// TwinCAT 3 PLC project Server
// ProgramVersion: 3.1.0.9
// libraries:
//   VisuElem3DPath, 3.5.6.0 (System)
//   VisuElemMeter, 3.5.6.0 (System)
//   VisuElems, 3.5.6.10 (System)
//   VisuElemsDateTime, 3.5.6.0 (System)
//   VisuElemsSpecialControls, 3.5.6.0 (System)
//   VisuElemsWinControls, 3.5.6.0 (System)
//   VisuElemTextEditor, 3.5.6.0 (System)
//   visuinputs, 3.5.6.0 (system)
//   VisuNativeControl, 3.5.6.0 (System)
//   Tc2_EtherCAT, * (Beckhoff Automation GmbH)
//   Tc2_Standard, * (Beckhoff Automation GmbH)
//   Tc2_System, * (Beckhoff Automation GmbH)
//   Tc2_Utilities, * (Beckhoff Automation GmbH)
//   Tc3_Interfaces, * (Beckhoff Automation GmbH)
//   Tc3_Module, * (Beckhoff Automation GmbH)
// project tree:
//   DUTs/ TUhr.TcDUT
//   / GlobalTextList.TcGTLO, PlcTask.TcTTO, Visualisiserungsmanager.TcVMO (not stored)
//   GVLs/ GVL.TcGVL, GVL_Constants.TcGVL, GVL_Visu.TcGVL, Haus1.TcGVL, Haus2.TcGVL, Haus4.TcGVL, HausSim.TcGVL, Netzwerk.TcGVL
//   Images/ Icons.TcIPO (not stored), ImagePool.TcIPO (not stored)
//   POUs/ FB_Alarm_Bild.TcPOU, FB_Alarm.TcPOU, FB_Besucher.TcPOU, FB_DataHistory_Int.TcPOU, FB_DataHistory_Real.TcPOU, FB_Heizung.TcPOU, FB_Regenmacher.TcPOU, FB_Uhr.TcPOU, FB_Visu_BildToggle.TcPOU, FB_Wetterbericht.TcPOU, FB_Wind.TcPOU, GET_TIME.TcPOU, INT_R_TRIG.TcPOU, MAIN.TcPOU, FB_Sonne.TcPOU, PG_Besucher.TcPOU, PG_Sonne.TcPOU, PG_Heizung.TcPOU, PG_Regen.TcPOU, PG_Simulationshaus.TcPOU, PG_Time.TcPOU, PG_Alarm.TcPOU, INT_TRIG.TcPOU, PG_Wind.TcPOU, PG_Visu.TcPOU, Visu_Baum.TcPOU, Visu_DayNight.TcPOU
//   VISUs/ Haus_1.TcVIS, Haus_2.TcVIS, Haus_3.TcVIS, MainVisu.TcVIS, Simuliertes_Haus.TcVIS, Settings.TcVIS, Uhr.TcVIS, Wetterbericht.TcVIS, Zentrale.TcVIS
// real-time tasks:
//   TASK PlcTask: cycle T#10ms, priority 20, ADS port 350
// I/O:
//   DEVICE Netzvariablen (EtherCAT Automation Protocol) (disabled), AmsNetId 192.168.252.131.2.1
//     Server (Publisher)
//     Haus_01
//     Haus_02
//     Haus_04
// variable links:
//   Server/Server Instance <-> Netzvariablen (EtherCAT Automation Protocol)/Haus_01
//     PlcTask Inputs/Netzwerk.net_alarm_01 <-> net_alarm_01/Inputs/VarData
//     PlcTask Inputs/Netzwerk.net_besucher_01 <-> net_besucher_01/Inputs/VarData
//     PlcTask Inputs/Netzwerk.net_heizung_01 <-> net_heizung_01/Inputs/VarData
//     PlcTask Inputs/Netzwerk.net_licht_01 <-> net_licht_01/Inputs/VarData
//   Server/Server Instance <-> Netzvariablen (EtherCAT Automation Protocol)/Haus_02
//     PlcTask Inputs/Netzwerk.net_alarm_02 <-> net_alarm_02/Inputs/VarData
//     PlcTask Inputs/Netzwerk.net_besucher_02 <-> net_besucher_02/Inputs/VarData
//     PlcTask Inputs/Netzwerk.net_heizung_02 <-> net_heizung_02/Inputs/VarData
//     PlcTask Inputs/Netzwerk.net_licht_02 <-> net_licht_02/Inputs/VarData
//   Server/Server Instance <-> Netzvariablen (EtherCAT Automation Protocol)/Haus_04
//     PlcTask Inputs/Netzwerk.net_alarm_04 <-> net_alarm_04/Inputs/VarData
//     PlcTask Inputs/Netzwerk.net_besucher_04 <-> net_besucher_04/Inputs/VarData
//     PlcTask Inputs/Netzwerk.net_heizung_04 <-> net_heizung_04/Inputs/VarData
//     PlcTask Inputs/Netzwerk.net_licht_04 <-> net_licht_04/Inputs/VarData
//   Server/Server Instance <-> Netzvariablen (EtherCAT Automation Protocol)/Server (Publisher)
//     PlcTask Outputs/Netzwerk.net_einbruch_alarm <-> net_einbruch_alarm/Outputs/VarData
//     PlcTask Outputs/Netzwerk.net_heizung_out <-> net_heizung/Outputs/VarData
//     PlcTask Outputs/Netzwerk.net_regen <-> net_regen/Outputs/VarData
//     PlcTask Outputs/Netzwerk.net_reset_besucher <-> net_reset_besucher/Outputs/VarData
//     PlcTask Outputs/Netzwerk.net_sonne <-> net_sonne/Outputs/VarData
//     PlcTask Outputs/Netzwerk.net_wind <-> net_wind/Outputs/VarData

CONFIGURATION Server
    RESOURCE PLC ON TwinCAT3
        TASK PlcTask(INTERVAL := T#10ms, PRIORITY := 20);
        PROGRAM MAIN WITH PlcTask : MAIN;
    END_RESOURCE
END_CONFIGURATION

// ---- DUTs/TUhr.TcDUT
TYPE TUhr :
STRUCT
	Stunde : REAL;
	Minute : REAL;
	Sekunde : REAL;
END_STRUCT
END_TYPE

// ---- GVLs/GVL.TcGVL
VAR_GLOBAL
	Alarm_H1_V : BOOL;
	Alarm_H2_V : BOOL;
	Alarm_H4_V : BOOL;
	
	Licht : INT;
	Regen : BOOL;
	SimZeitMultiplikator : INT;
	RealtimeManipulator : INT := RealtimeManipulator_STD;

	SimTagesFortschritt : REAL;
	SimMilliSekunde : INT;
	SimSekunde : INT;
	SimMinute : INT;
	SimStunde : INT;
	
	RealMilliSekunde : INT;
	RealSekunde : INT;
	RealMinute : INT;
	RealStunde : INT;
	
	SimRealTagSeitStart : INT;
	RealTagSeitStart : INT;
	
	SonneHistory : ARRAY [0..DatenHistoryZaehler] OF INT;
	WindHistory : ARRAY [0..DatenHistoryZaehler] OF REAL;
	
	Wind_V : INT;
	Wind_Auto : BOOL;
	Wind_Auto_V : BOOL;
	BWind : BOOL;
	
	Sonne_Auto : BOOL;
	Sonne_Auto_V : BOOL;
	Sonne_V	: INT;
	Sonne_A	: INT;
	L_Sonnenstand : INT;
	L_Sonne : STRING;
	L_Himmel : DWORD;
	L_Baum : INT;
	
	GL_Besucher : INT;
	GL_Besucher_reset : BOOL;
	GL_Alarm_reset : BOOL;
	GL_Besucher_reset_A : BOOL;
	
	Regenwahrscheinlichkeit : INT := Regenwahrscheinlichkeit_STD;
END_VAR

// ---- GVLs/GVL_Constants.TcGVL
VAR_GLOBAL CONSTANT
	
	DatenHistoryZaehler : INT := 50;
	Licht_min : INT := 100;
	Licht_max : INT := 2500;
	Alarm_time : TIME := T#10S;
	Heizung_reaktion : TIME := T#20S;
	Maximum_Wind : REAL := 300;
	BildMond : STRING := 'Mond';
	BildSonne : STRING := 'Sonne';
	BildEinbruchAlarm : STRING := 'Einbruch_rot';
	BildEinbruchOk : STRING := 'Einbruch_grun';
	BildRegen : STRING := 'Regen';
	BildWolke : STRING := 'Wolke';
	BildLicht : STRING := 'Licht';
	BildDunkel : STRING := 'Dunkel';
	ICON_Mond : STRING := 'ICON_Mond';
	ICON_Sonne : STRING := 'ICON_Sonne';
	ICON_Wolke : STRING := 'ICON_Wolke';
	ICON_Regen : STRING := 'ICON_Regen';
	ICON_WindRegen : STRING := 'ICON_WindRegen';
	ICON_WindWolke : STRING := 'ICON_WindWolke';
	
	RealtimeManipulator_STD : INT := 0;	
	Regenwahrscheinlichkeit_STD : INT := 30;
	TagNachtFixGrad : INT := -90;
	TagNachtMaxTransparenz : INT := 255;
END_VAR

// ---- GVLs/GVL_Visu.TcGVL
VAR_GLOBAL
	Rege_Heute : BOOL;
	RegenSimStunde : INT;
	RegenSimMinute : INT;
	Regen_Dauer : INT;
	RegenSimStunde_Ende : INT;
	RegenSimMinute_Ende : INT;
	
	Wetterbericht_Bild : STRING;
	Wetterbericht_Vorhersage_Bild: STRING;
	
	Simulation : BOOL := FALSE;
	
	
	Uhr : TUhr;
	
END_VAR

// ---- GVLs/Haus1.TcGVL
VAR_GLOBAL
	// Einbruchbild
	L_EinbruchBild : STRING;
	// Bild der Wolke (Wetter)
	WetterBild : STRING := BildWolke;
	// Bild Licht (Im Haus)
	BildLicht : STRING := GVL_Constants.BildLicht;
END_VAR

// ---- GVLs/Haus2.TcGVL
VAR_GLOBAL
	L_EinbruchBild : STRING;
	WetterBild : STRING := BildWolke;
	BildLicht : STRING := GVL_Constants.BildLicht;
END_VAR

// ---- GVLs/Haus4.TcGVL
VAR_GLOBAL
	L_EinbruchBild : STRING;
	WetterBild : STRING := BildWolke;
	BildLicht : STRING := GVL_Constants.BildLicht;
END_VAR

// ---- GVLs/HausSim.TcGVL
VAR_GLOBAL
	// Licht brennt
	L_Licht : BOOL;
	// Licht einschalten (Visu)
	L_Licht_V : BOOL;
	// Einbruchbild (Wechset)
	L_EinbruchBild : STRING;
	// Bild der Wolke
	WetterBild : STRING := BildWolke;
	// Bild Licht im Haus
	BildLicht : STRING := GVL_Constants.BildLicht;
	
	// Besucher zähler
	Besucher : INT;
	// Hat alarm
	Alarm : BOOL;
	// Alarm eingeschalten
	Alarm_V : BOOL;
	// Heizung Simulation
	heizung_SIM : INT;
	
	// Klingeln (Visu)
	Sim_Haus_Glocke : BOOL;
	// Alarm einschalten (Visu)
	Sim_Haus_Alarm : BOOL;
	// Alarm zurücksetzen (Haus Visu)
	Sim_Haus_ResetAlarm: BOOL;
END_VAR

// ---- GVLs/Netzwerk.TcGVL
VAR_GLOBAL
// Licht im Haus 1
	net_licht_01 AT %I* : BOOL;
// Licht im Haus 2
	net_licht_02 AT %I* : BOOL;
// Licht im Haus 4
	net_licht_04 AT %I* : BOOL;
// Besucher im Haus 1
	net_besucher_01 AT %I* : INT;
// Besucher im Haus 2
	net_besucher_02 AT %I* : INT;
// Besucher im Haus 4
	net_besucher_04 AT %I* : INT;
// Alarm im Haus 1
	net_alarm_01 AT %I* : BOOL;
// Alarm im Haus 2
	net_alarm_02 AT %I* : BOOL;
// Alarm im Haus 4
	net_alarm_04 AT %I* : BOOL;
// Heizung im Haus 1
	net_heizung_01 AT %I* : INT;
// Heizung im Haus 2
	net_heizung_02 AT %I* : INT;
// Heizung im Haus 4
	net_heizung_04 AT %I* : INT;


// Globaler Alarm
	net_einbruch_alarm AT %Q* : BOOL;
// Globale Besucher reset
	net_reset_besucher AT %Q* : BOOL;
// Simulierter Wind
	net_wind AT %Q* : REAL;
// Simulierter Regen
	net_regen AT %Q* : BOOL;
// Simuliertes Licht
	net_sonne AT %Q* : REAL;
// Heizung resultat
	net_heizung_out AT %Q* : INT;
END_VAR

// ---- POUs/MAIN.TcPOU
PROGRAM MAIN
VAR
END_VAR

PG_Time();
PG_Alarm();
PG_Sonne();
PG_Regen();
PG_Heizung();
PG_Wind();
PG_Visu();
PG_Besucher();
PG_SimulationsHaus();

END_PROGRAM

// ---- POUs/PG_Time.TcPOU
PROGRAM PG_Time
VAR
	FAKE_TIME: GET_TIME;
	REAL_TIME: GET_TIME;
	FB_Uhr_0: FB_Uhr;
END_VAR

REAL_TIME(_speed := RealtimeManipulator); // GET_TIME
Fake_Time(_speed := SimZeitMultiplikator); // GET_TIME
SimTagesFortschritt := Fake_Time._prog;
RealMilliSekunde := REAL_TIME._ms;
SimMilliSekunde := Fake_Time._ms;
RealSekunde := REAL_TIME._s;
SimSekunde := Fake_Time._s;
RealMinute := REAL_TIME._m;
SimMinute := Fake_Time._m;
RealStunde := REAL_TIME._h;
SimStunde := Fake_Time._h;
RealTagSeitStart := REAL_TIME._days;
SimRealTagSeitStart := Fake_Time._days;
FB_Uhr_0(_h := SimStunde, _min := SimMinute, _s := SimSekunde); // FB_Uhr
Uhr.Stunde := FB_Uhr_0.deg_h;
Uhr.Minute := FB_Uhr_0.deg_min;
Uhr.Sekunde := FB_Uhr_0.deg_s;

END_PROGRAM

// ---- POUs/GET_TIME.TcPOU
FUNCTION_BLOCK GET_TIME
VAR_INPUT
	_speed : INT;
END_VAR
VAR_OUTPUT
	_prog : REAL;
	_ms : INT;
	_s : INT;
	_m : INT;
	_h : INT;
	_days : INT;
END_VAR
VAR
	systemTime : GETSYSTEMTIME;
	firstH : BOOL := TRUE;
	ms_count : UDINT;
END_VAR

// Systemzeit auslesen und in Millisekunden, Sekunden, Minuten, Stunden sowie den Tagesfrotschritt in % berechnen.
systemTime();
ms_count := systemTime.timeLoDW / 10000;
ms_count := ms_count * LREAL_TO_UDINT(EXPT(10, _speed));
_ms  := UDINT_TO_INT(ms_count MOD 1000);
_s := UDINT_TO_INT((ms_count / 1000) MOD 60);
_m := UDINT_TO_INT((ms_count / 60000) MOD 60); 
_h := UDINT_TO_INT(((ms_count / 3600000) MOD 24));
_prog := 360 * DINT_TO_REAL(_h * 3600000 + (_m+1) * 60000 + (_s+1) * 1000 + _ms) / UDINT_TO_REAL(24 * 3600000);

// Tage seit Systemstart zählen
IF _h MOD 24 = 0 THEN
	IF firstH THEN
		_days := _days + 1;
		firstH := FALSE;
	END_IF
ELSE
	firstH := TRUE;
END_IF

END_FUNCTION_BLOCK

// ---- POUs/FB_Uhr.TcPOU
FUNCTION_BLOCK FB_Uhr
VAR_INPUT
	_h : INT;
	_min : INT;
	_s : INT;
END_VAR
VAR_OUTPUT
	deg_h : REAL;
	deg_min : REAL;
	deg_s : REAL;
END_VAR
VAR
	History : ARRAY[0..2] OF INT;
END_VAR

IF History[0] <> _h THEN
	History[0] := _h;
	deg_h := 30 * _h;
END_IF
IF History[1] <> _min THEN
	History[1] := _min;
	deg_min := _min * 6;
END_IF
IF History[2] <> _s THEN
	History[2] := _s;
	deg_s := _s * 6;
END_IF

END_FUNCTION_BLOCK

// ---- POUs/PG_Alarm.TcPOU
PROGRAM PG_Alarm
VAR
	Alarm_Off_Time: TIME := GVL_CONSTANTS.Alarm_time;
	Alarm_0: FB_Alarm;
	Alarm_Bild: FB_Alarm_Bild;
END_VAR

Alarm_0(
    AL_H1 := net_alarm_01,
    AL_H1_V := Alarm_H1_V,
    AL_H2 := net_alarm_02,
    AL_H2_V := Alarm_H2_V,
    AL_H4 := net_alarm_04,
    AL_H4_V := Alarm_H4_V,
    Al_Sim := HausSim.Alarm,
    Simulation := Simulation,
    T_Alarm := Alarm_Off_Time,
    reset := GL_Alarm_reset); // FB_Alarm
net_einbruch_alarm := Alarm_0.GL_Alarm;
Alarm_Bild(
    alarm := net_einbruch_alarm,
    h1Alarm := net_alarm_01,
    h2Alarm := net_alarm_02,
    h4Alarm := net_alarm_04,
    hSimAlarm := HausSim.Alarm,
    Bild_Alarm := BildEinbruchAlarm,
    BIld_Ok := BildEinbruchOk); // FB_Alarm_Bild
Haus1.L_EinbruchBild := Alarm_Bild.SH1;
Haus2.L_EinbruchBild := Alarm_Bild.SH2;
Haus4.L_EinbruchBild := Alarm_Bild.SH4;
HausSim.L_EinbruchBild := Alarm_Bild.SHSim;

END_PROGRAM

// ---- POUs/FB_Alarm.TcPOU
FUNCTION_BLOCK FB_Alarm
VAR_INPUT
	AL_H1 : BOOL;	
	AL_H1_V : BOOL;
	AL_H2 : BOOL;
	AL_H2_V : BOOL;
	AL_H4 : BOOL;
	AL_H4_V : BOOL;
	Al_Sim : BOOL;
	Simulation : BOOL;
	T_Alarm : TIME;
	reset : BOOL;
END_VAR
VAR_OUTPUT
	GL_Alarm : BOOL;
END_VAR
VAR
	HatAlarm : BOOL;
	Alarm_On : TOF;
	Trig : F_TRIG;
	Alarm : RS;
END_VAR

IF Simulation THEN
HatAlarm := 
	AL_H1 OR 
	AL_H2 OR 
	AL_H4 OR 
	AL_H1_V OR 
	AL_H2_V OR 
	AL_H4_V OR
	AL_Sim;
ELSE
	HatAlarm := 
	AL_H1 OR 
	AL_H2 OR 
	AL_H4 OR 
	AL_H1_V OR 
	AL_H2_V OR 
	AL_H4_V;
END_IF
	
Alarm_On(IN := HatAlarm, PT := T_Alarm);
TRIG(CLK := Alarm_On.Q);
Alarm(SET := HatAlarm, RESET1 :=  TRIG.Q OR reset, Q1 => GL_Alarm);

END_FUNCTION_BLOCK

// ---- POUs/FB_Alarm_Bild.TcPOU
FUNCTION_BLOCK FB_Alarm_Bild
VAR_INPUT
	alarm : BOOL;
	h1Alarm : BOOL;
	h2Alarm : BOOL;
	h4Alarm : BOOL;
	hSimAlarm : BOOL;
	Bild_Alarm : STRING;
	BIld_Ok : STRING;
END_VAR
VAR_OUTPUT
	SH1 : STRING;
	SH2 : STRING;
	SH4 : STRING;
	SHSim : STRING;
END_VAR
VAR
	first : BOOL := TRUE;
	RTrig_H1 : R_TRIG;
	RTrig_H2 : R_TRIG;
	RTrig_H4 : R_TRIG;
	RTrig_HSim : R_TRIG;
	FTrig_H1 : F_TRIG;
	FTrig_H2 : F_TRIG;
	FTrig_h4 : F_TRIG;
	FTrig_HSim : F_TRIG;
END_VAR

RTrig_H1(CLK := h1Alarm);
FTrig_H1(CLK := h1Alarm);
RTrig_H2(CLK := h1Alarm);
FTrig_H2(CLK := h1Alarm);
RTrig_H4(CLK := h1Alarm);
FTrig_H4(CLK := h1Alarm);
FTrig_HSim(CLK := hSimAlarm);
RTrig_HSim(CLK := hSimAlarm);

IF first THEN
	IF h1Alarm THEN
		SH1 := Bild_Alarm;
	ELSE
		SH1 := Bild_Ok;
	END_IF
	IF h2Alarm THEN
		SH2 := Bild_Alarm;
	ELSE
		SH2 := Bild_Ok;
	END_IF
	IF h4Alarm THEN
		SH4 := Bild_Alarm;
	ELSE
		SH4 := Bild_Ok;
	END_IF
	IF hSimAlarm THEN
		SHSim := Bild_Alarm;
	ELSE
		SHSIM := Bild_Ok;
	END_IF
	
first := FALSE;

ELSE
	IF RTRIG_H1.Q THEN
		SH1 := Bild_Alarm;
	ELSIF FTRIG_H1.Q THEN
		SH1 := Bild_Ok;
	END_IF
	IF RTRIG_H2.Q THEN
		SH2 := Bild_Alarm;
	ELSIF FTRIG_H2.Q THEN
		SH2 := Bild_Ok;
	END_IF
	IF RTRIG_H4.Q THEN
		SH4 := Bild_Alarm;
	ELSIF FTRIG_H4.Q THEN
		SH4 := Bild_Ok;
	END_IF
	IF RTRIG_HSIM.Q THEN
		SHSIM := Bild_Alarm;
	ELSIF FTRIG_HSim.Q THEN
		SHSim := Bild_Ok;
	END_IF
END_IF

END_FUNCTION_BLOCK

// ---- POUs/PG_Sonne.TcPOU
PROGRAM PG_Sonne
VAR
	Sun_history: FB_DataHistory_Int;
	INT_TRIG_0: INT_TRIG;
	FB_Sonne_1: FB_Sonne;
	R_TRIG_0: R_TRIG;
END_VAR
VAR // added by the converter: edge detectors and wires of the graphical bodies
    _w1 : BOOL;
END_VAR

R_TRIG_0(CLK := Sonne_Auto_V); // R_TRIG
_w1 := R_TRIG_0.Q XOR _w1;
Sonne_Auto := NOT _w1;
FB_Sonne_1(
    _val := SimTagesFortschritt,
    _auto := Sonne_Auto,
    _visu_val := Sonne_V,
    _time := RealSekunde,
    _min := Licht_min,
    _max := Licht_max); // FB_Sonne
Licht := FB_Sonne_1._sin;
Sun_history(_val := FB_Sonne_1._sin, _save := FB_Sonne_1._trig); // FB_DataHistory_Int
SonneHistory := Sun_history._array;
net_sonne := REAL_TO_INT(Licht);

END_PROGRAM

// ---- POUs/FB_DataHistory_Int.TcPOU
FUNCTION_BLOCK FB_DataHistory_Int
VAR_INPUT
	_val : INT;
	_save : BOOL;
END_VAR
VAR_OUTPUT
	_array : ARRAY [0..DatenHistoryZaehler] OF INT;
END_VAR
VAR
	_i : INT;
END_VAR

IF _save THEN
	FOR _i := 0 TO DatenHistoryZaehler - 1 DO
		_array[_i] := _array[_i + 1];
	END_FOR
	_array[DatenHistoryZaehler] := _val;
END_IF

END_FUNCTION_BLOCK

// ---- POUs/INT_TRIG.TcPOU
FUNCTION_BLOCK INT_TRIG
VAR_INPUT
	_val : INT;
END_VAR
VAR_OUTPUT
	_Q : BOOL;
END_VAR
VAR
	History : INT;
	first : BOOL := TRUE;
END_VAR

// R_Trig und F_Trig in einem für INT Werte.
IF first THEN
	History := _val;
	first := FALSE;
ELSE
	IF History <> _val THEN
		_Q := TRUE;
		History := _val;
	ELSIF _Q THEN
		_Q := FALSE;	
	END_IF
END_IF

END_FUNCTION_BLOCK

// ---- POUs/FB_Sonne.TcPOU
FUNCTION_BLOCK FB_Sonne
VAR CONSTANT
	dayFix : INT := -90;
END_VAR
VAR_INPUT
	_val : REAL;
	_auto : BOOL;
	_visu_val : INT;
	_time : INT;
	_min : INT;
	_max : INT;
END_VAR
VAR_OUTPUT
	_sin : INT;
	_trig : BOOL;
END_VAR
VAR
	_do : BOOL;
	diff : INT;
	average : INT;
	T_Trig : INT_Trig;
END_VAR

// Trigger für die Ausführung alle 1sek.
T_Trig(_val := _time, _Q => _do);
// _do wird für die History (Statistik) verwendet.
_trig := _do;


// Wenn Licht Automatik eingeschalten, Automatisch berechnen
IF _do AND _auto THEN
	// Berechnen der Lichtemmission anhand der Uhrzeit _val
	diff := (_max - _min) / 2;
	average := REAL_TO_INT(_min + diff);
	_sin := LREAL_TO_INT(SIN(DEG_TO_RAD(_val + dayFix)) * diff + average);
ELSIF _do THEN
	// Wenn Licht Automatik ausgeschalten, Wert von Slider nehmen.
	_sin := _visu_val;
END_IF

END_FUNCTION_BLOCK

// ---- POUs/PG_Regen.TcPOU
PROGRAM PG_Regen
VAR
	Regenmacher: FB_Regenmacher;;
	Wetterbericht: FB_Wetterbericht;
END_VAR
VAR // added by the converter: edge detectors and wires of the graphical bodies
    _w1 : ANY;
END_VAR

Regenmacher(
    _gen := Regenwahrscheinlichkeit <> 0,
    _m := SimMinute,
    _h := SimStunde,
    _day := SimRealTagSeitStart,
    _prozent := Regenwahrscheinlichkeit,
    Simulation := TRUE); // FB_Regenmacher
Regen := Regenmacher._rain;
Rege_Heute := Regenmacher.HeuteRegen;
RegenSimStunde := Regenmacher.RegenStunde;
RegenSimMinute := Regenmacher.RegenMinute;
Regen_Dauer := Regenmacher.RegenDauer;
RegenSimStunde_Ende := Regenmacher.RegenBisStunde;
RegenSimMinute_Ende := Regenmacher.RegenBisMinute;
_w1 := SEL(Regen, BildWolke, BildRegen);
Haus1.WetterBild := _w1;
Haus2.WetterBild := _w1;
Haus4.WetterBild := _w1;
HausSim.WetterBild := _w1;
Wetterbericht(Regen := Regen, Wind := net_wind > 0); // FB_Wetterbericht
Wetterbericht_Bild := Wetterbericht.Aktuell;
Wetterbericht_Vorhersage_Bild := Wetterbericht.Vorhersage;

END_PROGRAM

// ---- POUs/FB_Regenmacher.TcPOU
FUNCTION_BLOCK FB_Regenmacher
VAR_INPUT
	_gen : BOOL;
	_m : INT;
	_h : INT;
	_day : INT;
	_prozent : INT;
	Simulation : BOOL;
END_VAR
VAR_OUTPUT
	_rain : BOOL;
	HeuteRegen : BOOL;
	RegenStunde : INT;
	RegenMinute : INT;
	RegenDauer : INT;
	RegenBisStunde : INT;
	RegenBisMinute : INT;
END_VAR
VAR
	dayTrig : INT_R_TRIG;
	RAND_H : DRAND;
	RAND_M : DRAND;
	RAND_D : DRAND;
END_VAR

IF _gen AND Simulation THEN
	dayTrig(_val := _day);
	
	IF dayTrig._Q THEN
		_rain := FALSE;
		HeuteRegen := FALSE;
		RAND_H(Seed := 0);
		HeuteRegen := LREAL_TO_INT(RAND_H.Num * 100) < _prozent;
		
		IF HeuteRegen THEN
			RAND_M(Seed := 1);
			RAND_D(Seed := 2);
			RegenStunde := LREAL_TO_INT(RAND_H.Num * 12);
			RegenMinute := LREAL_TO_INT(RAND_M.Num * 59);
			RegenDauer := LREAL_TO_INT(RAND_D.Num * 480);
			RegenBisStunde := RegenStunde + (RegenDauer / 60);
			RegenBisMinute := RegenMinute + (RegenDauer - ((RegenBisStunde - RegenStunde) * 60));
			IF RegenBisMinute > 60 THEN
				RegenBisStunde := RegenBisStunde + 1;
				RegenBisMinute := RegenBisMinute - 60;
			END_IF
		END_IF
	END_IF
	
	IF HeuteRegen THEN
		IF RegenStunde < _h OR (RegenStunde = _h AND RegenMinute <= _m) THEN
			_rain := TRUE;
			IF RegenBisStunde <= _h AND RegenBisMinute <= _m THEN
				_rain := FALSE;
				HeuteRegen := FALSE;
			END_IF
		END_IF
	END_IF
ELSE
	_rain := FALSE;
	HeuteRegen := FALSE;
END_IF

END_FUNCTION_BLOCK

// ---- POUs/INT_R_TRIG.TcPOU
FUNCTION_BLOCK INT_R_TRIG
VAR_INPUT
	_val : INT;
END_VAR
VAR_OUTPUT
	_Q : BOOL;
END_VAR
VAR
	History : INT;
	first : BOOL := TRUE;
END_VAR

// R_Trig für INT Werte. 
IF first THEN
	History := _val;
	first := FALSE;
ELSE
	IF History < _val THEN
		_Q := TRUE;
		History := _val;
	ELSIF _Q THEN
		_Q := FALSE;	
	END_IF
END_IF

END_FUNCTION_BLOCK

// ---- POUs/FB_Wetterbericht.TcPOU
FUNCTION_BLOCK FB_Wetterbericht
VAR_INPUT
	Regen : BOOL;
	Wind : BOOL;
	HeuteRegen : BOOL;
END_VAR
VAR_OUTPUT
	Aktuell : STRING;
	Vorhersage : STRING;
END_VAR
VAR
END_VAR

// Das richtige Icon anzeigen anhand der Wetterbedingungen
IF Regen AND Wind THEN
	Aktuell := GVL_CONSTANTS.ICON_WindRegen;
ELSIF Regen THEN
	Aktuell := GVL_CONSTANTS.ICON_Regen;
ELSIF Wind THEN
	Aktuell := GVL_CONSTANTS.ICON_WindWolke;
ELSE
	Aktuell := GVL_CONSTANTS.ICON_Wolke;
END_IF

IF HeuteRegen THEN
	Vorhersage := GVL_CONSTANTS.ICON_Regen;
ELSE
	Vorhersage := GVL_CONSTANTS.ICON_Wolke;
END_IF

END_FUNCTION_BLOCK

// ---- POUs/PG_Heizung.TcPOU
PROGRAM PG_Heizung
VAR
	FB_Heizung_0: FB_Heizung;
END_VAR

FB_Heizung_0(
    Heizung_01 := net_heizung_01,
    Heizung_02 := net_heizung_02,
    Heizung_04 := net_heizung_04,
    Heizung_Sim := HausSim.heizung_SIM,
    Simulation := Simulation,
    react := Heizung_reaktion); // FB_Heizung
net_heizung_out := FB_Heizung_0.Heizung;

END_PROGRAM

// ---- POUs/FB_Heizung.TcPOU
FUNCTION_BLOCK FB_Heizung
VAR_INPUT
	Heizung_01 : INT;
	Heizung_02 : INT;
	Heizung_04 : INT;
	Heizung_Sim : INT;
	Simulation : BOOL;
	react : TIME;
END_VAR
VAR_OUTPUT
	Heizung : INT;
END_VAR
VAR
	history : ARRAY [0..4] OF INT;
	first : BOOL := TRUE;
	_i : INT;
	maximum : INT := 0;
	timer : TON;
	
	run_timer : BOOL := FALSE;
END_VAR

IF FIRST THEN
	history[0] := Heizung_01;
	history[1] := Heizung_02;
	history[2] := Heizung_04;
	IF Simulation THEN
		history[3] := Heizung_Sim;
	ELSE
		history[3] := 0;
	END_IF
	
	FOR _i := 0 TO 3 DO
		IF history[_i] > maximum THEN
			maximum := history[_i];
		END_IF
	END_FOR
	history[4] := maximum;
	IF maximum < 15 THEN
		Heizung := 15;
	ELSIF maximum > 30 THEN
		Heizung := 30;
	ELSE
		Heizung := maximum;
	END_IF

	FIRST := FALSE;
ELSE
	// Wen es eine Änderung der Werte gab (Sim Haus nur miteinbeziehen, wenn Simulation eingeschalten ist.
	IF history[0] <> Heizung_01 OR history[1] <> Heizung_02 OR history[2] <> Heizung_04 OR (history[3] <> Heizung_Sim AND Simulation) THEN
		history[0] := Heizung_01;
		history[1] := Heizung_02;
		history[2] := Heizung_04;
		
		IF Simulation THEN
			history[3] := Heizung_Sim;
		ELSE
			history[3] := 0;
		END_IF
		
		// Höchsten Wert finden
		FOR _i := 0 TO 3 DO
			IF history[_i] > maximum THEN
				maximum := history[_i];
			END_IF
		END_FOR
		// Prüfen ob Wert ungleich beim Letzen mal und Timer starten bis neue Temperatur gesendet wird
		IF maximum <> history[4] THEN
			run_timer := TRUE;
			history[4] := maximum;	
		END_IF
	END_IF
END_IF

// Sendeverzögerung der neuen Temperatur.
IF run_timer THEN
	IF timer.Q THEN
		run_timer := FALSE;
		IF history[4] < 15 THEN
			Heizung := 15;
		ELSIF history[4] > 30 THEN
			Heizung := 30;
		ELSE
			Heizung := history[4];
		END_IF
	END_IF
	timer(IN := run_timer, PT := react);
END_IF

END_FUNCTION_BLOCK

// ---- POUs/PG_Wind.TcPOU
PROGRAM PG_Wind
VAR
	FB_Wind_0: FB_Wind;
	INT_TRIG_0: INT_TRIG;
	FB_DataHistory_Real_0: FB_DataHistory_Real;
	R_TRIG_0: R_TRIG;
END_VAR
VAR // added by the converter: edge detectors and wires of the graphical bodies
    _w1 : BOOL;
END_VAR

R_TRIG_0(CLK := Wind_Auto_V); // R_TRIG
_w1 := R_TRIG_0.Q XOR _w1;
Wind_Auto := NOT _w1;
FB_Wind_0(_auto := Wind_auto, _wind_V := Wind_V, _max := GVL_Constants.Maximum_Wind, _time := RealSekunde); // FB_Wind
net_wind := FB_Wind_0.Wind;
FB_DataHistory_Real_0(_val := FB_Wind_0.Wind, _save := FB_Wind_0.Trig); // FB_DataHistory_Real
WindHistory := FB_DataHistory_Real_0._array;
BWInd := net_wind > 0;

END_PROGRAM

// ---- POUs/FB_Wind.TcPOU
FUNCTION_BLOCK FB_Wind
VAR_INPUT
	_auto : BOOL;
	_wind_V : INT;
	_max : REAL;
	_time : INT;
END_VAR
VAR_OUTPUT
	Wind : REAL := 0;
	Trig : BOOL;
END_VAR
VAR
	Count : INT := 0;
	speed : REAL := 0.01;
	Step : BOOL := TRUE;
	valToAdd : REAL;
	
	StartTime : TON;
	StopTime : TON;
	NoWind : TP;
	NoWindFirst : BOOL := TRUE;
	StartT : TIME := T#2S;
	StopT : TIME := T#2S;
	Rand : DRAND;
	Direction : BOOL := TRUE;
	Prog : REAL;
	Height : REAL := 100;
	T_Trig : INT_Trig;
	_do : BOOL;
	_manipulator : INT := 100;
	WindToZero : REAL;
	BWindToZero : BOOL := FALSE;
 END_VAR

StartTime(IN := Direction, PT := StartT);
StopTime(IN := NOT Direction, PT := StopT);
T_TRIG(_val := _time, _Q => _do);
NoWind(IN := count = 0, PT := T#30S);

Trig := _do;

IF NoWind.Q THEN
	_do := FALSE;
	Wind := 0;
END_IF

IF _do AND _auto THEN
	IF Direction THEN
		Prog := ( TIME_TO_REAL(StartTime.ET) / TIME_TO_REAL(StartT) ) * 90 ;
		IF StartTime.Q THEN
			Direction := FALSE;
			Rand();
			StopT := LREAL_TO_TIME(Rand.Num * 10000);
			count := count + 1;
		END_IF
	ELSE
		IF count = 7 THEN
			WindToZero := Wind;
			BWindToZero := TRUE;
		END_IF
		
		Prog := 90 - ( TIME_TO_REAL(StopTime.ET) / TIME_TO_REAL(StopT) ) * 90;
		
		IF StopTime.Q THEN
				Direction := TRUE;
				Rand();
				StartT := LREAL_TO_TIME(Rand.Num * 10000);
				Step := NOT STEP;
				IF count = 7 THEN
					count := 0;
					BWindToZero := FALSE;
				ELSE
					count := count + 1;
				END_IF
			END_IF
	END_IF	

	IF count = 7 AND BWindToZero THEN
		Wind := WindToZero * LREAL_TO_REAL(SIN(DEG_TO_RAD(Prog)));
	ELSE
		valToAdd := LREAL_TO_REAL(SIN(DEG_TO_RAD(Prog)) * (TIME_TO_REAL(StartT) / _manipulator) ) ;
			
		IF STEP THEN
			valToAdd := valToAdd * ((_max - Wind) / _max);
			Wind := WIND + valToAdd;
		ELSE
			valToAdd := valToAdd * (Wind / _max);
			Wind := WIND - valToAdd;
		END_IF
	END_IF
END_IF

IF NOT _auto THEN
	Wind := _wind_V;
END_IF

END_FUNCTION_BLOCK

// ---- POUs/FB_DataHistory_Real.TcPOU
FUNCTION_BLOCK FB_DataHistory_Real
VAR_INPUT
	_val : REAL;
	_save : BOOL;
END_VAR
VAR_OUTPUT
	_array : ARRAY [0..DatenHistoryZaehler] OF REAL;
END_VAR
VAR
	_i : INT;
END_VAR

IF _save THEN
	FOR _i := 0 TO DatenHistoryZaehler - 1 DO
		_array[_i] := _array[_i + 1];
	END_FOR
	_array[DatenHistoryZaehler] := _val;
END_IF

END_FUNCTION_BLOCK

// ---- POUs/PG_Visu.TcPOU
PROGRAM PG_Visu
VAR
	Visu_Baum_0: Visu_Baum;
	INT_TRIG_0: INT_TRIG;
	Visu_DayNight_0: Visu_DayNight;
	INT_TRIG_1: INT_TRIG;
	BildToggle_Haus1: FB_Visu_BildToggle;
	BildToggle_Haus2: FB_Visu_BildToggle;
	BildToggle_Haus4: FB_Visu_BildToggle;
	BildToggle_HausSim: FB_Visu_BildToggle;
END_VAR
VAR // added by the converter: edge detectors and wires of the graphical bodies
    _w1 : ANY;
END_VAR

BildToggle_HausSim(val := HausSim.L_Licht, s_t := GVL_Constants.BildLicht, s_f := GVL_Constants.BildDunkel); // FB_Visu_BildToggle
BildToggle_Haus4(s_t := GVL_Constants.BildLicht, s_f := GVL_Constants.BildDunkel); // FB_Visu_BildToggle
Haus1.BildLicht := BildToggle_Haus1.BILD;
BildToggle_Haus2(val := net_licht_02, s_t := GVL_Constants.BildLicht, s_f := GVL_Constants.BildDunkel); // FB_Visu_BildToggle
INT_TRIG_1(_val := SimSekunde / 10); // INT_TRIG
Haus2.BildLicht := BildToggle_Haus2.BILD;
Haus4.BildLicht := BildToggle_Haus4.BILD;
HausSim.BildLicht := BildToggle_HausSim.BILD;
_w1 := (INT_TRIG_1._Q OR INT_TRIG_0._Q) AND BWind;
INT_TRIG_0(_val := SimMilliSekunde / 10); // INT_TRIG
Visu_Baum_0(_rotate := _w1, _speed := 1, _minDeg := -20, _maxDeg := 20); // Visu_Baum
L_Baum := Visu_Baum_0._rot;
Visu_DayNight_0(_deg := SimTagesFortschritt, licht := Licht, Licht_min := Licht_min, Licht_max := Licht_max); // Visu_DayNight
L_Sonne := Visu_DayNight_0._day;
L_Sonnenstand := Visu_DayNight_0._stand;
L_Himmel := Visu_DayNight_0._sun;
BildToggle_Haus1(val := net_licht_01, s_t := GVL_Constants.BildLicht, s_f := GVL_Constants.BildDunkel); // FB_Visu_BildToggle
// net_licht_04: input not connected

END_PROGRAM

// ---- POUs/Visu_Baum.TcPOU
FUNCTION_BLOCK Visu_Baum
VAR_INPUT
_rotate : BOOL;	
_speed : INT;
_minDeg : INT := -90;
_maxDeg : INT := 90;
END_VAR
VAR_OUTPUT
	_rot : INT := 0;
END_VAR
VAR
	counter : INT;
	rotateRight : BOOL;
END_VAR

// Wenn es Windet, bewegt sich der Baum.
IF _rotate THEN
	IF rotateRight THEN
		IF _rot > _maxDeg THEN
			rotateRight := FALSE;
		ELSE
			_rot := _rot + _speed;
		END_IF
	ELSE
		IF _rot < _minDeg THEN
			rotateRight := TRUE;
		ELSE
			_rot := _rot - _speed;
		END_IF
	END_IF
END_IF

END_FUNCTION_BLOCK

// ---- POUs/Visu_DayNight.TcPOU
FUNCTION_BLOCK Visu_DayNight
VAR CONSTANT
	Fix_Degree : INT := GVL_Constants.TagNachtFixGrad;
END_VAR
VAR_INPUT
	_deg : REAL;
	licht : INT;
	Licht_min : INT;
	Licht_max : INT;
END_VAR
VAR_OUTPUT
	_day : STRING;
	_stand : INT;
	_sun : DWORD;
END_VAR
VAR
	timeProg : REAL;
	transparency : INT := GVL_Constants.TagNachtMaxTransparenz;
	color : STRING;
	HEX : STRING;
END_VAR

timeProg := _deg + Fix_Degree;
IF timeProg < 0 OR timeProg > 180 THEN
	_stand := REAL_TO_INT(timeProg + 180);
	_day := GVL_Constants.BildMond;
ELSE
	_day := GVL_Constants.BildSonne;
	_stand := REAL_TO_INT(timeProg);
END_IF

transparency := REAL_TO_INT( ((Licht - Licht_min) / INT_TO_REAL(Licht_max - Licht_min)) * GVL_Constants.TagNachtMaxTransparenz );

HEX := DWORD_TO_HEXSTR(INT_TO_UINT(transparency), 2, FALSE);

color := '16#';
color := CONCAT(color, HEX);
color := CONCAT(color, 'FFFF00');

_sun := STRING_TO_DWORD(color);

END_FUNCTION_BLOCK

// ---- POUs/FB_Visu_BildToggle.TcPOU
FUNCTION_BLOCK FB_Visu_BildToggle
VAR_INPUT
	val : BOOL;
	s_t : STRING;
	s_f : STRING;
END_VAR
VAR_OUTPUT
	BILD : STRING;
END_VAR
VAR
	FIRST : BOOL := TRUE;
	history : BOOL;
END_VAR

// Selectorbaustein um einen String (Bild ID) Zumzuschalten
IF FIRST THEN
	IF val THEN
		BILD := s_t;
	ELSE
		BILD := s_f;
	END_IF
	history := val;
END_IF

IF val <> history THEN
	IF val THEN
		BILD := s_t;
	ELSE
		BILD := s_f;
	END_IF
	history := val;
END_IF

END_FUNCTION_BLOCK

// ---- POUs/PG_Besucher.TcPOU
PROGRAM PG_Besucher
VAR
	FB_Besucher_0: FB_Besucher;
	INT_R_TRIG_0: INT_R_TRIG;
END_VAR

INT_R_TRIG_0(_val := SimRealTagSeitStart); // INT_R_TRIG
GL_Besucher_reset_A := INT_R_TRIG_0._Q;
FB_Besucher_0(
    bes_H1 := net_besucher_01,
    bes_H2 := net_besucher_02,
    bes_H4 := net_besucher_04,
    bes_Sim := HausSim.Besucher,
    Simulation := Simulation,
    res_V := GL_Besucher_reset,
    res_A := GL_Besucher_reset_A); // FB_Besucher
GL_Besucher := FB_Besucher_0.besucher;
net_reset_besucher := FB_Besucher_0.res;

END_PROGRAM

// ---- POUs/FB_Besucher.TcPOU
FUNCTION_BLOCK FB_Besucher
VAR_INPUT
	bes_H1 : INT;
	bes_H2 : INT;
	bes_H4 : INT;
	bes_Sim : INT;
	Simulation : BOOL;
	res_V : BOOL;
	res_A : BOOL;
END_VAR
VAR_OUTPUT
	besucher : INT;
	res : BOOL;
END_VAR
VAR
END_VAR

IF Simulation THEN
	besucher := bes_H1 + bes_H2 + bes_H4 + bes_Sim;
ELSE
	besucher := bes_H1 + bes_H2 + bes_H4;
END_IF
IF res_V OR res_A THEN
	res := TRUE;
ELSE
	res := FALSE;
END_IF

END_FUNCTION_BLOCK

// ---- POUs/PG_Simulationshaus.TcPOU
PROGRAM PG_Simulationshaus
VAR
	Besucher: CTU;
	RS_0: RS;
	R_TRIG_0: R_TRIG;
	R_TRIG_1: R_TRIG;
END_VAR
VAR // added by the converter: edge detectors and wires of the graphical bodies
    _w1, _w2 : BOOL;
END_VAR

Besucher(CU := Sim_Haus_Glocke, RESET := net_reset_besucher); // CTU
HausSim.Besucher := WORD_TO_INT(Besucher.CV);
R_TRIG_0(CLK := HausSim.Alarm_V); // R_TRIG
_w1 := R_TRIG_0.Q XOR _w1;
HausSim.Alarm := _w1;
R_TRIG_1(CLK := HausSim.L_Licht_V); // R_TRIG
_w2 := R_TRIG_1.Q XOR _w2;
HausSim.L_Licht := _w2;

END_PROGRAM

// ---- GlobalTextList.TcGTLO
TEXTLIST GlobalTextList
  68 = ''
  26 = '%10i'
  15 = '%10s'
  1 = '%2f'
  2 = '%2i'
  4 = '%2i : '
  3 = '%2i : %2i : %2i'
  13 = '%2i Lumen'
  28 = '%2i Regenwahrscheinlichkeit'
  11 = '%2i Tage '
  10 = '%2i Tge '
  9 = '%2ih'
  8 = '%2imin'
  6 = '%2ims'
  7 = '%2is'
  62 = '%2r km/h Wind'
  5 = '%i'
  30 = '%i %'
  51 = '%i : Heizung'
  63 = '%i km/h Wind'
  66 = '%i Lumen'
  29 = '%i Regenwahrscheinlichkeit'
  14 = '%s'
  37 = 'Aktuelles Wetter'
  18 = 'Alarm'
  21 = 'Alarm %b'
  57 = 'Alarm zurücksetzen'
  67 = 'asdf'
  16 = 'Besucher'
  17 = 'Besucher Hochzählen'
  56 = 'Besucher zurücksetzen'
  55 = 'Besucher zurücksetzen%i'
  22 = 'Besucher: %i'
  54 = 'Besucher: %i°C'
  20 = 'Besuchern'
  48 = 'Den ganzen Tag schönes Wetter'
  35 = 'Einstellungen'
  50 = 'Globaler Alarm'
  31 = 'Haus 1'
  32 = 'Haus 2'
  33 = 'Haus 4'
  19 = 'Heizung'
  24 = 'Heizung: %2i'
  25 = 'Heizung: %2r'
  23 = 'Heizung: %i'
  52 = 'Heizung: %i°C'
  59 = 'Licht'
  12 = 'Real Time'
  45 = 'Regen bis: %i'
  49 = 'Regen Dauer: %i'
  69 = 'Regen Dauer: %i min'
  41 = 'Regen um: %i'
  42 = 'Regen um: %i Uhr'
  27 = 'Regenwahrscheinlichkeit'
  36 = 'Schliessen'
  47 = 'Schön bis: %i'
  34 = 'Settings'
  60 = 'Simulation'
  58 = 'Simulations Haus'
  64 = 'Sonne'
  65 = 'Sonne Manuell'
  46 = 'Uhr %i'
  44 = 'Uhr und %i Minuten'
  43 = 'und %i Minuten'
  38 = 'Vorhersage'
  39 = 'Vorhersage  Heute'
  40 = 'Vorhersage Heute'
  61 = 'Wind Manuell'
  53 = 'Wind: %i'
  0 = 'Zeit Manipulation'
END_TEXTLIST

// ---- VISUs/Haus_1.TcVIS
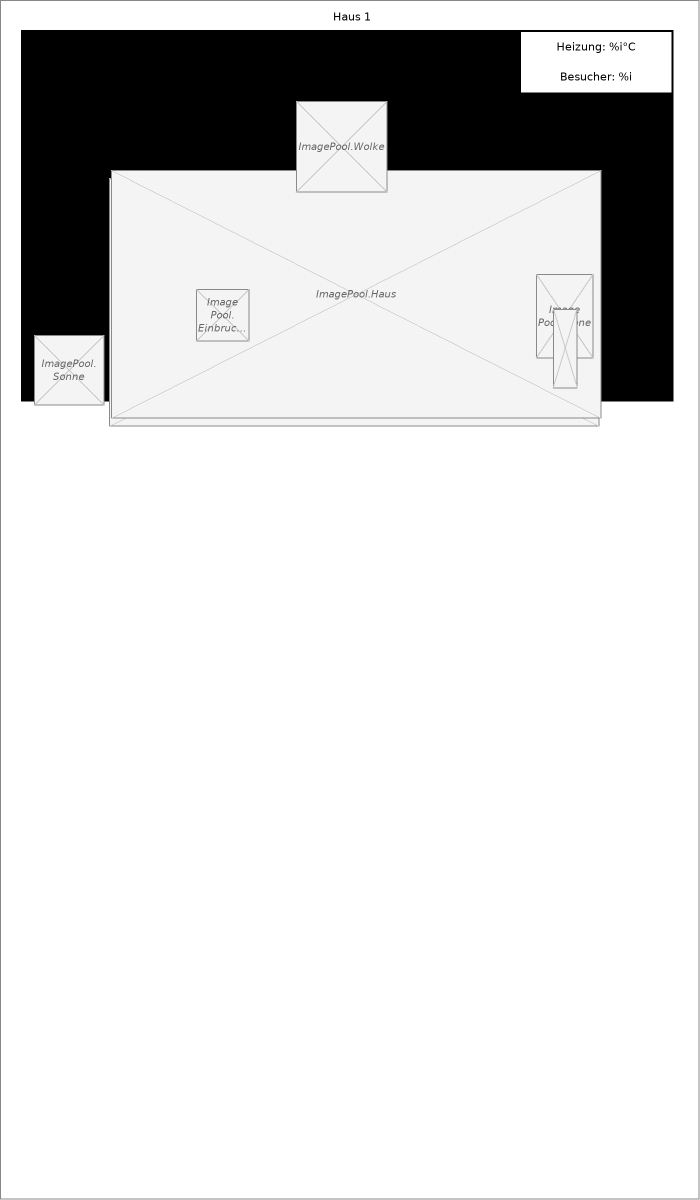
VISUALIZATION Haus_1  // 700x1200
    Rectangle (21,30 652x371)
    Rectangle (21,30 652x371), colour variable: L_Himmel
        p2167032090: L_Himmel
    Image (109,178 490x248), image: ImagePool.Licht
        p84334746: Haus1.BildLicht
    Image (111,170 490x248), image: ImagePool.Haus
    Image (536,274 57x84), image: ImagePool.Krone
        p2858320360: L_Baum
    Image (553,309 24x79), image: ImagePool.Stamm
    Image (34,335 70x70), image: ImagePool.Sonne
        p2858320360: L_Sonnenstand
        p84334746: L_Sonne
    Image (196,289 53x52), image: ImagePool.Einbruch_grun
        p84334746: Haus1.L_EinbruchBild
    Image (296,101 91x91), image: ImagePool.Wolke
        p84334746: Haus1.WetterBild
    Textfield (277,6 150x22), "Haus 1"
    Textfield (521,32 150x30), "Heizung: %i°C", text variable: net_heizung_01
    Textfield (521,62 150x30), "Besucher: %i", text variable: net_besucher_01
END_VISUALIZATION

// ---- VISUs/Haus_2.TcVIS
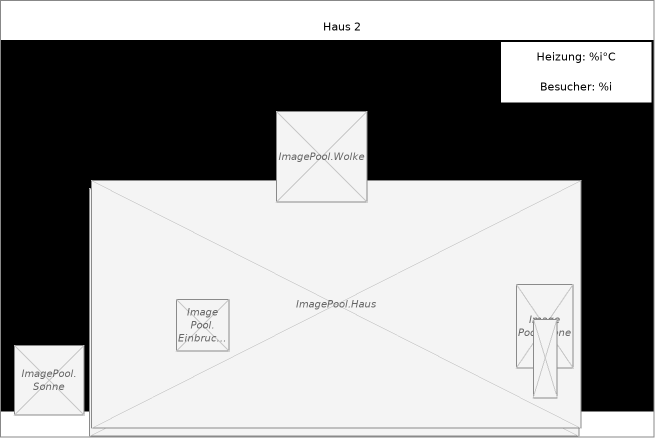
VISUALIZATION Haus_2  // 655x438
    Rectangle (1,40 652x371)
    Rectangle (1,40 652x371), colour variable: L_Himmel
        p2167032090: L_Himmel
    Image (89,188 490x248), image: ImagePool.Licht
        p84334746: Haus2.BildLicht
    Image (91,180 490x248), image: ImagePool.Haus
    Image (516,284 57x84), image: ImagePool.Krone
        p2858320360: L_Baum
    Image (533,319 24x79), image: ImagePool.Stamm
    Image (14,345 70x70), image: ImagePool.Sonne
        p2858320360: L_Sonnenstand
        p84334746: L_Sonne
    Image (176,299 53x52), image: ImagePool.Einbruch_grun
        p84334746: Haus2.L_EinbruchBild
    Image (276,111 91x91), image: ImagePool.Wolke
        p84334746: Haus2.WetterBild
    Textfield (267,16 150x22), "Haus 2"
    Textfield (501,42 150x30), "Heizung: %i°C", text variable: net_heizung_02
    Textfield (501,72 150x30), "Besucher: %i", text variable: net_besucher_02
END_VISUALIZATION

// ---- VISUs/Haus_3.TcVIS
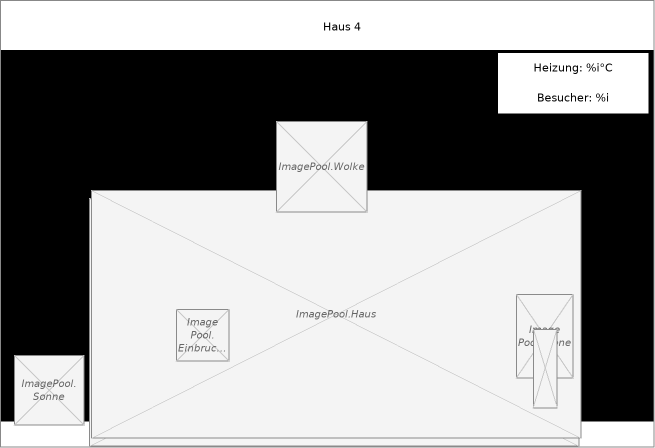
VISUALIZATION Haus_3  // 655x448
    Rectangle (1,50 652x371)
    Rectangle (1,50 652x371), colour variable: L_Himmel
        p2167032090: L_Himmel
    Image (89,198 490x248), image: ImagePool.Licht
        p84334746: Haus4.BildLicht
    Image (91,190 490x248), image: ImagePool.Haus
    Image (516,294 57x84), image: ImagePool.Krone
        p2858320360: L_Baum
    Image (533,329 24x79), image: ImagePool.Stamm
    Image (14,355 70x70), image: ImagePool.Sonne
        p2858320360: L_Sonnenstand
        p84334746: L_Sonne
    Image (176,309 53x52), image: ImagePool.Einbruch_grun
        p84334746: Haus4.L_EinbruchBild
    Image (276,121 91x91), image: ImagePool.Wolke
        p84334746: Haus4.WetterBild
    Textfield (267,16 150x22), "Haus 4"
    Textfield (498,53 150x30), "Heizung: %i°C", text variable: net_heizung_04
    Textfield (498,83 150x30), "Besucher: %i", text variable: net_besucher_04
END_VISUALIZATION

// ---- VISUs/MainVisu.TcVIS
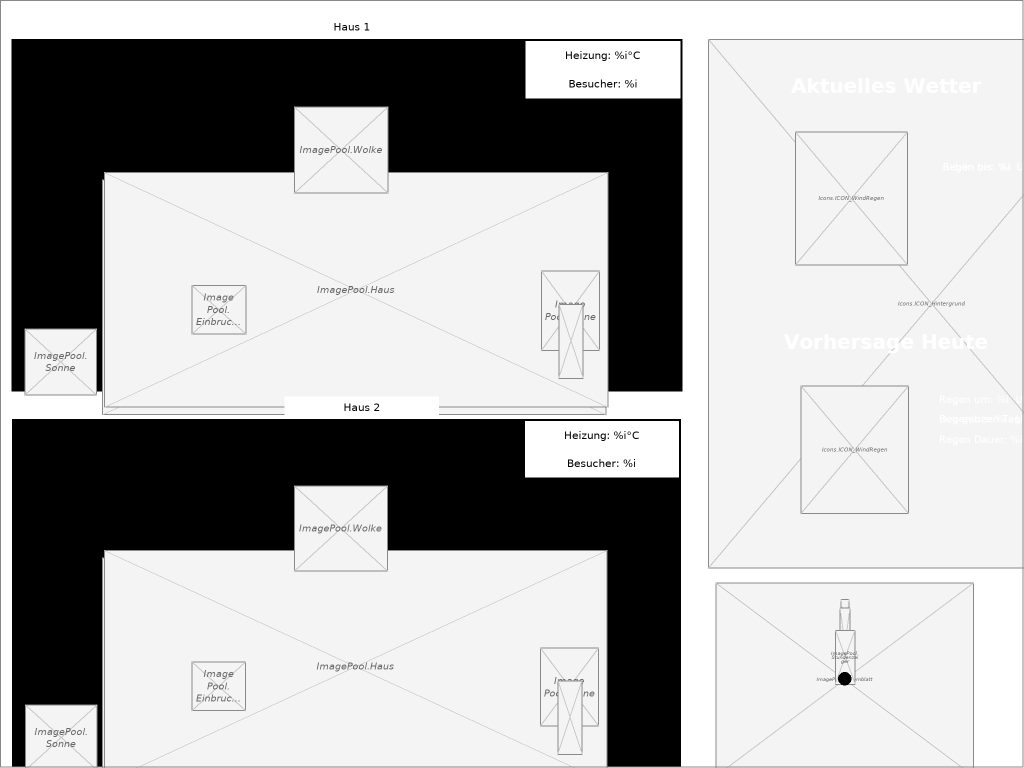
VISUALIZATION MainVisu  // 1024x768
    Frame (-10,11 720x1138), frame switch variable: Simulation
        shows Haus_1()
        shows Simuliertes_Haus()
    Frame (8,754 678x410), invisible if: Simulation
        shows Haus_3()
    Frame (11,382 672x410), invisible if: Simulation
        shows Haus_2()
    Button (1325,51 150x30), "Settings"
        OnMouseClick: OpenDialog Dialog=Settings, OpenModal=True, OpenCentered=True
    Frame (709,39 572x508)
        shows Wetterbericht()
    Frame (713,819 291x209)
        shows Zentrale()
    Button (1327,112 150x30), "Simulation"
        toggle Simulation
        OnMouseClick: OpenDialog Dialog=Simuliertes_Haus, OpenModal=True, PositionX=50, PositionY=50
        OnMouseClick: CloseDialog Dialog=Simuliertes_Haus, Result=OK, NumpadKeypadSet=True
    Frame (736,574 226x226)
        shows Uhr()
END_VISUALIZATION

// ---- VISUs/Simuliertes_Haus.TcVIS
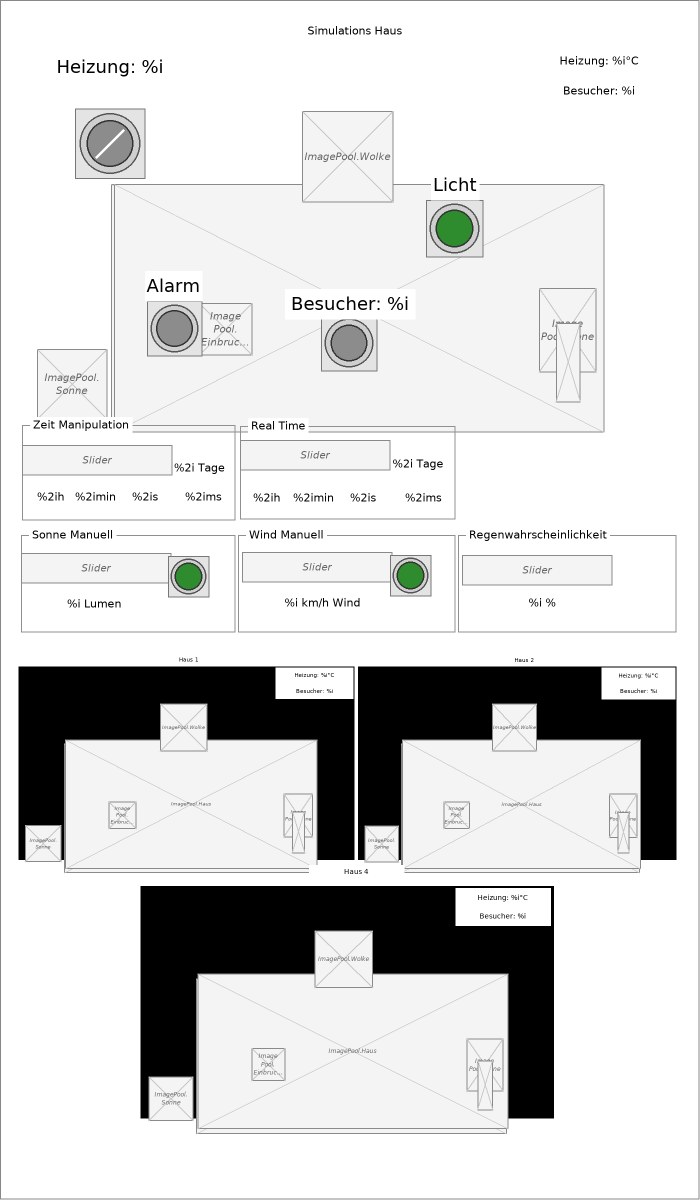
VISUALIZATION Simuliertes_Haus  // 700x1200
    Frame (8,651 360x625)
        shows Haus_1()
    Rectangle (24,44 652x371)
    Rectangle (24,44 652x371), colour variable: L_Himmel
        p2167032090: L_Himmel
    Image (111,184 490x248), image: ImagePool.Licht
        p84334746: HausSim.BildLicht
    Image (114,184 490x248), image: ImagePool.Haus
    Image (539,288 57x84), image: ImagePool.Krone
        p2858320360: L_Baum
    Image (556,323 24x79), image: ImagePool.Stamm
    Image (37,349 70x70), image: ImagePool.Sonne
        p2858320360: L_Sonnenstand
        p84334746: L_Sonne
    Image (199,303 53x52), image: ImagePool.Einbruch_grun
        p84334746: HausSim.L_EinbruchBild
    Image (302,111 91x91), image: ImagePool.Wolke
        p84334746: HausSim.WetterBild
    PushSwitch (147,300 55x57), variable: HausSim.Alarm_V, behaviour: TAP, style: Switch-PushSwitch-Gray
    Rectangle (145,271 57x30), "Alarm"
    Textfield (280,20 150x22), "Simulations Haus"
    Textfield (524,46 150x30), "Heizung: %i°C", text variable: HausSim.heizung_SIM
    Textfield (524,76 150x30), "Besucher: %i", text variable: HausSim.Besucher
    GroupBox (22,417 213x103), "Zeit Manipulation"
        Slider (0,28 150x30), variable: SimZeitMultiplikator, scale 0..4
        Textfield (41,65 65x30), "%2imin", text variable: SimMinute
        Textfield (90,65 66x30), "%2is", text variable: SimSekunde
        Textfield (148,65 67x30), "%2ims", text variable: SimMilliSekunde
        Textfield (-2,65 62x30), "%2ih", text variable: SimStunde
        Textfield (149,36 61x30), "%2i Tage", text variable: SimRealTagSeitStart
    PushSwitch (426,200 57x57), variable: HausSim.L_Licht_V, behaviour: TAP, style: Switch-PushSwitch-Green
    Rectangle (431,170 48x30), "Licht", text variable: HausSim.Besucher
    GroupBox (240,418 215x101), "Real Time"
        Textfield (149,31 62x30), "%2i Tage", text variable: RealTagSeitStart
        Slider (0,22 150x30), variable: RealtimeManipulator, scale 0..3
        Textfield (41,65 65x30), "%2imin", text variable: RealMinute
        Textfield (90,65 66x30), "%2is", text variable: RealSekunde
        Textfield (150,65 67x30), "%2ims", text variable: RealMilliSekunde
        Textfield (-4,65 62x30), "%2ih", text variable: RealStunde
    GroupBox (458,527 218x105), "Regenwahrscheinlichkeit"
        Slider (4,28 150x30), variable: Regenwahrscheinlichkeit, scale 0..100
        Textfield (-18,61 205x30), "%i %", text variable: Regenwahrscheinlichkeit
    GroupBox (238,527 217x105), "Wind Manuell"
        Slider (4,25 150x30), variable: Wind_V, scale 0..200
        Textfield (-18,61 205x30), "%i km/h Wind", text variable: net_wind
        PushSwitch (152,28 41x41), variable: Wind_Auto_V, behaviour: TAP, style: Switch-PushSwitch-Green
    GroupBox (21,527 214x105), "Sonne Manuell"
        Slider (0,26 150x30), variable: Sonne_V, scale 100..2500
        Textfield (4,62 139x30), "%i Lumen", text variable: net_sonne
        PushSwitch (147,29 41x41), variable: Sonne_Auto_V, behaviour: TAP, style: Switch-PushSwitch-Green
    Frame (358,646 319x228)
        shows Haus_2()
    Frame (140,855 415x280)
        shows Haus_3()
    PushSwitch (321,314 56x58), variable: Sim_Haus_Glocke, behaviour: TAP, style: Switch-PushSwitch-Gray
    Rectangle (285,289 130x30), "Besucher: %i", text variable: HausSim.Besucher
    Potentiometer360 (75,105 70x77), variable: heizung_SIM, style: Potentiometer-Potentiometer360-Gray, scale format: %.1f, scale 14..30
    Rectangle (35,52 150x30), "Heizung: %i", text variable: heizung_SIM
END_VISUALIZATION

// ---- VISUs/Settings.TcVIS
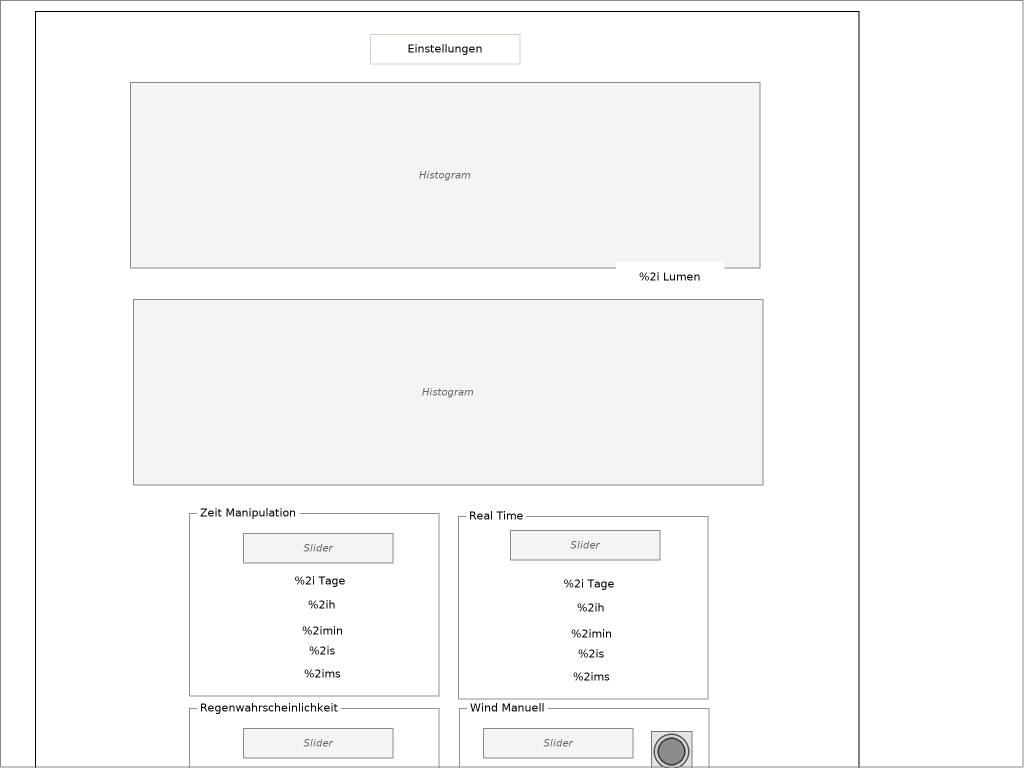
VISUALIZATION Settings  // 1024x768
    Rectangle (35,11 824x973)
    Histogram (130,82 630x186), scale format: %i, scale 0..3000
        p1518820177: SonneHistory
        p102497268: SonneHistory
        p788070771: ARRAY [0..DatenHistoryZaehler] OF INT
    GroupBox (189,505 250x191), "Zeit Manipulation"
        Slider (54,28 150x30), variable: SimZeitMultiplikator, scale 0..4
        Textfield (102,61 62x30), "%2i Tage", text variable: SimRealTagSeitStart
        Textfield (101,111 65x30), "%2imin", text variable: SimMinute
        Textfield (100,131 66x30), "%2is", text variable: SimSekunde
        Textfield (100,154 67x30), "%2ims", text variable: SimMilliSekunde
        Textfield (102,85 62x30), "%2ih", text variable: SimStunde
    GroupBox (458,508 250x191), "Real Time"
        Textfield (102,61 62x30), "%2i Tage", text variable: RealTagSeitStart
        Slider (52,22 150x30), variable: RealtimeManipulator, scale 0..3
        Textfield (101,111 65x30), "%2imin", text variable: RealMinute
        Textfield (100,131 66x30), "%2is", text variable: RealSekunde
        Textfield (100,154 67x30), "%2ims", text variable: RealMilliSekunde
        Textfield (102,85 62x30), "%2ih", text variable: RealStunde
    Textfield (616,262 108x30), "%2i Lumen", text variable: Licht
    GroupBox (189,700 250x105), "Regenwahrscheinlichkeit"
        Slider (54,28 150x30), variable: Regenwahrscheinlichkeit, scale 0..100
        Textfield (32,61 205x30), "%i %", text variable: Regenwahrscheinlichkeit
    Textfield (370,34 150x30), "Einstellungen"
    Button (680,929 150x30), "Schliessen"
        OnMouseClick: CloseDialog Dialog=Settings, Result=OK, NumpadKeypadSet=True
    Histogram (133,299 630x186), scale format: %i, scale 0..500
        p1518820177: WindHistory
        p102497268: WindHistory
        p788070771: ARRAY [0..DatenHistoryZaehler] OF REAL
    GroupBox (459,700 250x105), "Wind Manuell"
        Slider (24,28 150x30), variable: Wind_V, scale 0..200
        Textfield (2,61 205x30), "%i km/h Wind", text variable: net_wind
        PushSwitch (192,31 41x41), variable: Wind_Auto_V, behaviour: TAP, style: Switch-PushSwitch-Gray
    GroupBox (189,816 250x105), "Sonne Manuell"
        Slider (40,28 150x30), variable: Sonne_V, scale 100..2500
        Textfield (44,65 139x30), "%i Lumen", text variable: net_sonne
        PushSwitch (197,32 41x41), variable: Sonne_Auto_V, behaviour: TAP, style: Switch-PushSwitch-Gray
END_VISUALIZATION

// ---- VISUs/Uhr.TcVIS
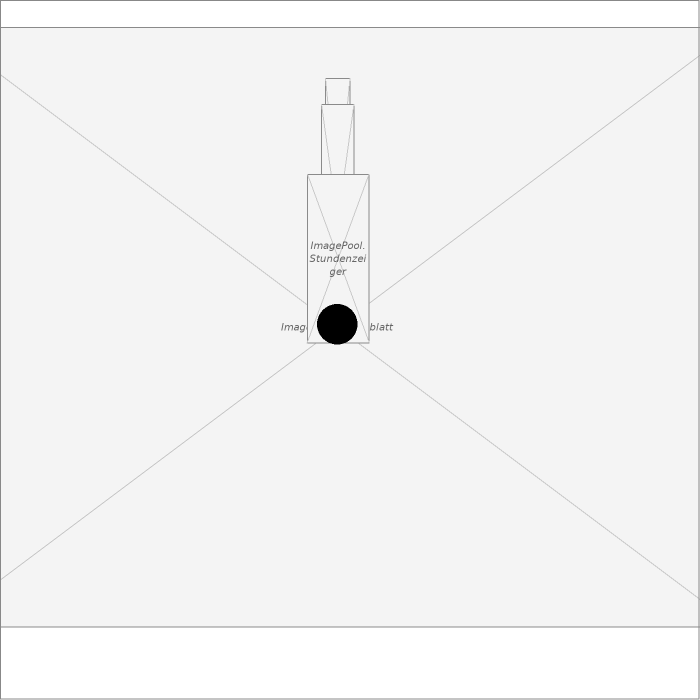
VISUALIZATION Uhr  // 700x700
    Image (-63,27 800x600), image: ImagePool.Ziffernblatt
    Image (325,78 25x260), image: ImagePool.Sekundenzeiger
        p2858320360: Uhr.Sekunde
    Image (321,104 33x239), image: ImagePool.Minutenzeiger
        p2858320360: Uhr.Minute
    Image (307,174 62x169), image: ImagePool.Stundenzeiger
        p2858320360: Uhr.Stunde
    Ellipse (317,304 40x40)
END_VISUALIZATION

// ---- VISUs/Wetterbericht.TcVIS
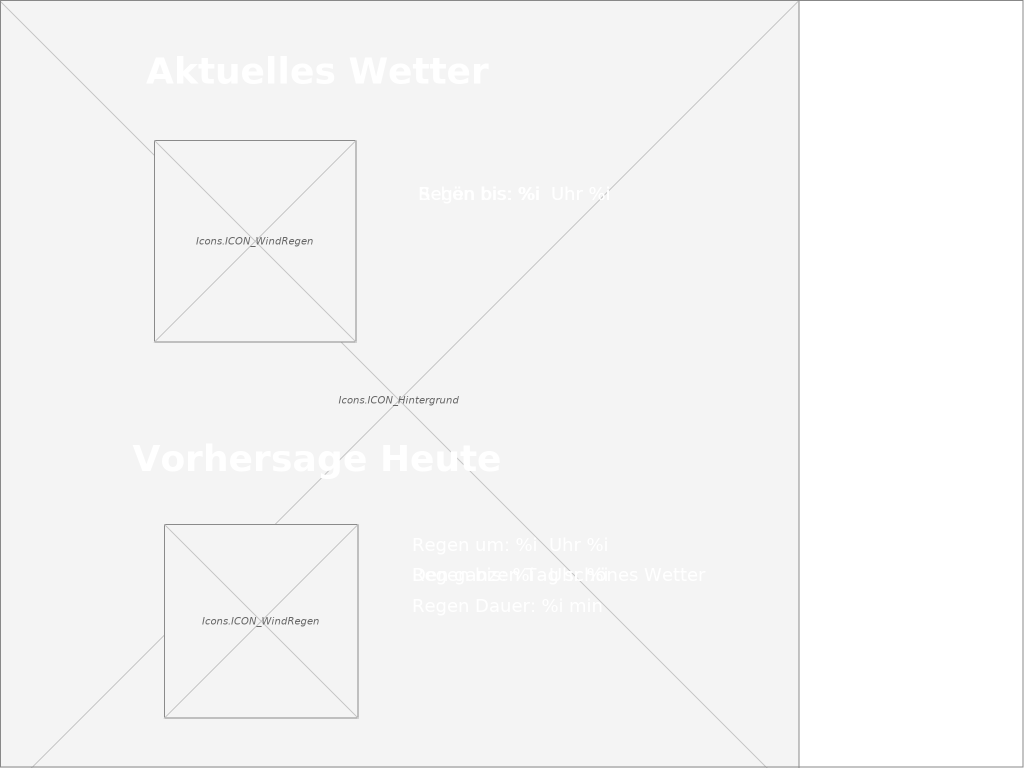
VISUALIZATION Wetterbericht  // 1024x768
    Image (-1,0 800x800), image: Icons.ICON_Hintergrund
    Image (154,140 202x202), image: Icons.ICON_WindRegen
        p84334746: Wetterbericht_Bild
    Label (121,56 393x30), "Aktuelles Wetter"
    Label (121,430 392x57), "Vorhersage Heute"
    Image (164,524 194x194), image: Icons.ICON_WindRegen
        p84334746: Wetterbericht_Vorhersage_Bild
    Textfield (409,530 231x30), "Regen um: %i", text variable: RegenSimStunde, invisible if: NOT Rege_Heute
    Textfield (546,530 231x30), "Uhr %i", text variable: RegenSimMinute, invisible if: NOT Rege_Heute
    Textfield (409,560 231x30), "Regen bis: %i", text variable: RegenSimStunde_Ende, invisible if: NOT Rege_Heute
    Textfield (546,560 231x30), "Uhr %i", text variable: RegenSimMinute_Ende, invisible if: NOT Rege_Heute
    Textfield (409,591 231x30), "Regen Dauer: %i min", text variable: Regen_Dauer, invisible if: NOT Rege_Heute
    Textfield (364,179 231x30), "Regen bis: %i", text variable: RegenSimStunde_Ende, invisible if: NOT Regen
    Textfield (548,179 231x30), "Uhr %i", text variable: RegenSimMinute_Ende, invisible if: NOT Regen
    Textfield (364,179 231x30), "Schön bis: %i", text variable: RegenSimStunde, invisible if: NOT Rege_Heute OR Regen
    Textfield (548,179 231x30), "Uhr %i", text variable: RegenSimMinute, invisible if: NOT Rege_Heute OR Regen
    Textfield (409,560 352x30), "Den ganzen Tag schönes Wetter", text variable: RegenSimStunde, invisible if: Rege_Heute
END_VISUALIZATION

// ---- VISUs/Zentrale.TcVIS
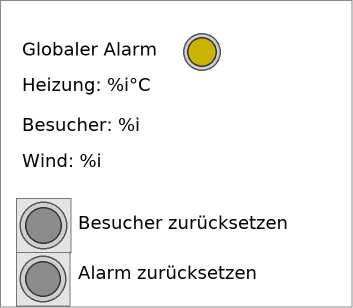
VISUALIZATION Zentrale  // 353x308
    Lamp1 (180,30 44x44), variable: net_einbruch_alarm, style: Lamp-Lamp1-Yellow
    Label (19,35 191x29), "Globaler Alarm"
    Textfield (19,70 150x30), "Heizung: %i°C", text variable: net_heizung_out
    Textfield (19,110 150x30), "Besucher: %i", text variable: GL_Besucher
    Textfield (19,146 150x30), "Wind: %i", text variable: net_wind
    PushSwitch (16,198 55x55), variable: GL_Besucher_reset, behaviour: TAP, style: Switch-PushSwitch-Gray
    PushSwitch (16,252 54x54), variable: GL_Alarm_reset, behaviour: TAP, style: Switch-PushSwitch-Gray
    Textfield (75,208 276x30), "Besucher zurücksetzen"
    Textfield (75,258 276x30), "Alarm zurücksetzen"
END_VISUALIZATION
